TYPE Selection :

	(All_Blinds ,Small_Wall, Big_Wall, Glass_Wall);

END_TYPE

(* stored: Version 1.1.0.1, ProductVersion 3.1.4024.12
   DUT Selection: Id {a73397a3-5b95-4c48-aadb-a088026b4c55} *)
